INTERFACE I_HeatCoolControl

METHOD SetTemperature
VAR_INPUT
	nSetTemperature	: UINT;
END_VAR
END_METHOD

END_INTERFACE

(* stored: Version 1.1.0.1, ProductVersion 3.1.4024.4
   Itf I_HeatCoolControl: Id {547de773-5a7a-4a26-bfa8-9bf9f4c2abaf}
   Method SetTemperature: Id {15d48f39-5425-405b-ac5b-ddd5e6b34968} *)
